INTERFACE ITF_Base

PROPERTY Definition : REFERENCE TO ST_BaseDefinition
GET
END_GET
END_PROPERTY

PROPERTY EnableManualControl : Bool
SET
END_SET
END_PROPERTY

END_INTERFACE

(* stored: Version 1.1.0.1
   Itf ITF_Base: Id {f927fc98-80f2-4c43-8ca7-3a1dc177fbb8}
   Property Definition: Id {d3f380f3-139f-4c79-9cc9-daf5cb03a0ef}
   Get Get: Id {406c1840-fb71-40c6-832d-088762f4eca3}
   Property EnableManualControl: Id {bd485c9d-33f4-40ef-a176-6d3e976ee598}
   Set Set: Id {78d70ea4-8243-4fa4-bacc-bc59f662c5dc} *)
